// TIA Portal V18 export
// export: Created 2025-12-01T17:52:57.7890867Z, ExportSetting None, DisplayName Totally Integrated Automation Portal, DisplayVersion V18 Update 5, DisplayName TIA Portal Openness, DisplayVersion V18 Update 5, DisplayName TIA Portal Teamcenter Gateway, DisplayVersion V18, DisplayName TIA Portal Version Control Interface, DisplayVersion V18, DisplayName STEP 7 Professional, DisplayVersion V18 Update 5, DisplayName STEP 7 Safety, DisplayVersion V18, DisplayName WinCC Professional, DisplayVersion V18 Update 5
Screen "215 X80Scanner_800A1"  1280x800, Number=215, Template=02ManualUnit1
  ScreenLayer "Layer_0"
    FaceplateInstance "RCS_fpKeyenceSR1000_TP1200_1" at 10,129 size 1134x421  FaceplateTypeName=KeyenceSR1000@$@03_FacePlate@$@RCS_fpKeyenceSR1000_TP1200 V 0.0.6
      InterfacePropertyText "文本"  Text="800A1_TableCodeScan"
      Property := KeyenceSR1000Ctrl_800A1DB_sHMI
    Button "btnMenu6_1" at 768,725 size 128x75  TextOff="A-读码器 800A1 / A-CodeReader 800A1", TextOn="A-读码器 800A1 / A-CodeReader 800A1"
      on Click: ActivateScreen(Screen name := , Object number := 0)
    Button "btnMenu4" at 384,725 size 128x75  TextOff="A-伺服 381A1 / A-Servo 381A1", TextOn="A-伺服 381A1 / A-Servo 381A1"
      on Click: ActivateScreen(Screen name := 212-Servo_381A1, Object number := 0)
    Button "btnMenu5" at 512,725 size 128x75  TextOff="A-读码器 801A1 / A-CodeReader 801A1", TextOn="A-读码器 801A1 / A-CodeReader 801A1"
      on Click: ActivateScreen(Screen name := 213 Scanner_801A1, Object number := 0)
    Button "btnMenu6" at 640,725 size 128x75  TextOff="A-读码器 804A1 / A-CodeReader 804A1", TextOn="A-读码器 804A1 / A-CodeReader 804A1"
      on Click: ActivateScreen(Screen name := 214 Scanner_804A1, Object number := 0)
    Button "btnMenu7" at 896,725 size 128x75
    Button "btnMenu7_1" at 1024,725 size 128x75  TextOff="下一页 / NextPage", TextOn="下一页 / NextPage"
      on Click: ActivateScreen(Screen name := 216_Cylinder_A2, Object number := 0)
    Button "btnMenu4_1" at 256,725 size 128x75  TextOff="A-伺服 380A1 / A-Servo 380A1", TextOn="A-伺服 380A1 / A-Servo 380A1"
      on Click: ActivateScreen(Screen name := 211-Servo_380A1, Object number := 0)
    Button "按钮_1" at 128,725 size 128x75  PictureOff=向右箭头_0, TextOff="A-气缸1 / A-Cylinder1", TextOn="A-气缸1 / A-Cylinder1"
      on Click: ActivateScreen(Screen name := 210_Cylinder_A1, Object number := 0)
